FUNCTION_BLOCK FB_HNLTMachineSystem
VAR_INPUT
END_VAR
VAR_OUTPUT
END_VAR
VAR
END_VAR

END_FUNCTION_BLOCK

(* stored: Version 1.1.0.1, ProductVersion 3.1.4024.10
   POU FB_HNLTMachineSystem: Id {9e31bb33-93a7-4fc1-a5d6-51b03d50941a}, SpecialFunc None *)
